Staubli VAL3: start.pgx

program start()
begin
  logMsg("RemoteControl - Version " + toString("", VERSION))

  call init()
  enablePower()

  // Move to the initial starting pose
  logMsg("[INIT] Moving dangerously to starting position")
  movej(BASE_POSE, mount, SLOW_CONFIG)
  waitEndMove()

  taskCreate TASK_NAMES["SocketHandler"], 5, socketHandler()
  taskCreate TASK_NAMES["MotionWorker"], 10, motionWorker()
  taskCreate TASK_NAMES["MotionSupervisor"], 20, motionSupervisor()
  taskCreate TASK_NAMES["MovingReporter"], 29, movingReporter()
  taskCreate TASK_NAMES["MotionReporter"], 30, motionReporter()
end
